{attribute 'qualified_only'}
// LREAL: Long Real decimal number

VAR_GLOBAL
	fPressureSupplyFiltered		: LREAL; 	// Filtered supply pressure
	fPressurePistonSideFiltered : LREAL; 	// Filtered pressure, piston side
	fPressureRodSideFiltered 	: LREAL; 	// Filtered pressure, rod side
	fValveOutputFiltered		: LREAL; 	// Filtered valve output
	fValveOutputUnfiltered		: LREAL; 	// Unfiltered valve output
	fPressurePaLower			: LREAL;  	// Filtered value before counterbalance valve
END_VAR

(* stored: Version 1.1.0.1
   GVL G_Filtered: Id {d9539014-b5a8-4af3-b695-54bf1cf81853} *)
